PROGRAM F15_CaseControlCACData_ORG
VAR
	rtrigScanBarcode				: R_TRIG;
	fbScannerCtrl					: FB_SCANNER_CameraSelect;
	bScanCaseLabel				: BOOL;
	fbCaseLableEvaluation			: FB_SCANNER_Evaluation;

	rtrigSetCaseValidationOK			: R_TRIG;
	rtrigSetCaseValidationNOK		: R_TRIG;

	sCaseSerialCode				: T_CASE_Barcode;
	sFirstOuterInCase				: T_OUTER_Barcode;
	sLastOuterInCase				: T_OUTER_Barcode;
	sFirstPackSerialCode			: T_PACK_Barcode;
	sLastPackSerialCode				: T_PACK_Barcode;


	fbSequenceControl				: FB_SYSTEM_SeqControl;
	nSequenceStep				: INT;
	b00_Idle						: BOOL;
	b01_ScanLabel					: BOOL;
	b03_CreateFileName			: BOOL;
	b05_MoveCaseData				: BOOL;
	b08_WriteFSSFile				: BOOL;
	b10_CaseTraceValid			: BOOL;
	b18_CaseValid					: BOOL;
	b19_CaseInvalid				: BOOL;
	b20_Done						: BOOL;

	bDone						: BOOL;
	bBusy						: BOOL;
	tonScanTimeout					: TON;
	tonOverTime				: TON;

	rtrigCACData				: R_TRIG;
	tF15TimeExecution		: TIME;
	bTestSeq						: BOOL;
	sCACFileTemplate				: T_CAC_Filename;

	stValidateCACData				: ST_CAC_Data;
	fbMoveCaseData				: FB_CASE_ValidateAndMoveCACData;

	sPrintCaseContent				: STRING(255);

	fbPopulateCHMData				: FB_CHM_PopulateDataForFSS3;
	fbWriteCHMFile				: FB_CHM_WriteFSS3Files; (*Old system supporting FSS2 -> FB_CHM_WriteFSSFile;*)

	fbWriteCACToArchive 			: FB_CAC_WriteToArchive_v2;
	fbWriteCACToArchiveDB			: FB_CAC_WriteHierachyToDB;
	fbCaseStatusPulse				: TON;
	bCACValid					: BOOL;
	bCHMValid					: BOOL;


	fbMoveVerifiedCAC				: FB_CASE_MoveVerifiedCAC;
	fbMoveFailedCAC				: FB_CASE_MoveFailedCAC;

	fbCaseEfficiency				: FB_KPI_GenericEfficiency;
	fbCaseInspectionEfficiency		: FB_KPI_CaseEfficiency;
	(*fbCaseInspectionEfficiency		: FB_KPI_PACAN_CaseEfficiency;*)
	fbRejectCount					: CTU;
	nRejectActualCount				: INT;

	fbCaseValidationScanned			: FB_CTU32;
	fbCaseValidationCorrect			: FB_CTU32;
	fbCaseValidationNoCaseLabel		: FB_CTU32;
	fbCaseValidationCasePackerReject	: FB_CTU32;

	aLastCaseBarcodes				: ARRAY[1..cMAX_LAST_CASE_BARCODES] OF T_CASE_Barcode;
	fbAddVerifiedCaseBarcode		: FB_CASE_AddVerifiedCaseBarcode;

	fbCaseLevelCounter	: FB_KPI_CaseLevelCounter;
	tofCaseValidationCameraOFFDelay 	: TOF;

	fbFileWriteCACError				: FB_LOG_FileWriteError;
	fbFileWriteCHMError			: FB_LOG_FileWriteError;

END_VAR
(*
VAR CONSTANT
	sOptions						: ST_SCANNER_Options := (eScannerType := E_MV_440SR_FULL, nImageBuffer := 1, nExpectedResp := 1);
END_VAR*)
VAR // added by the converter: edge detectors and wires of the graphical bodies
    _w1 : ANY;
    _w2, _w3 : BOOL;
END_VAR

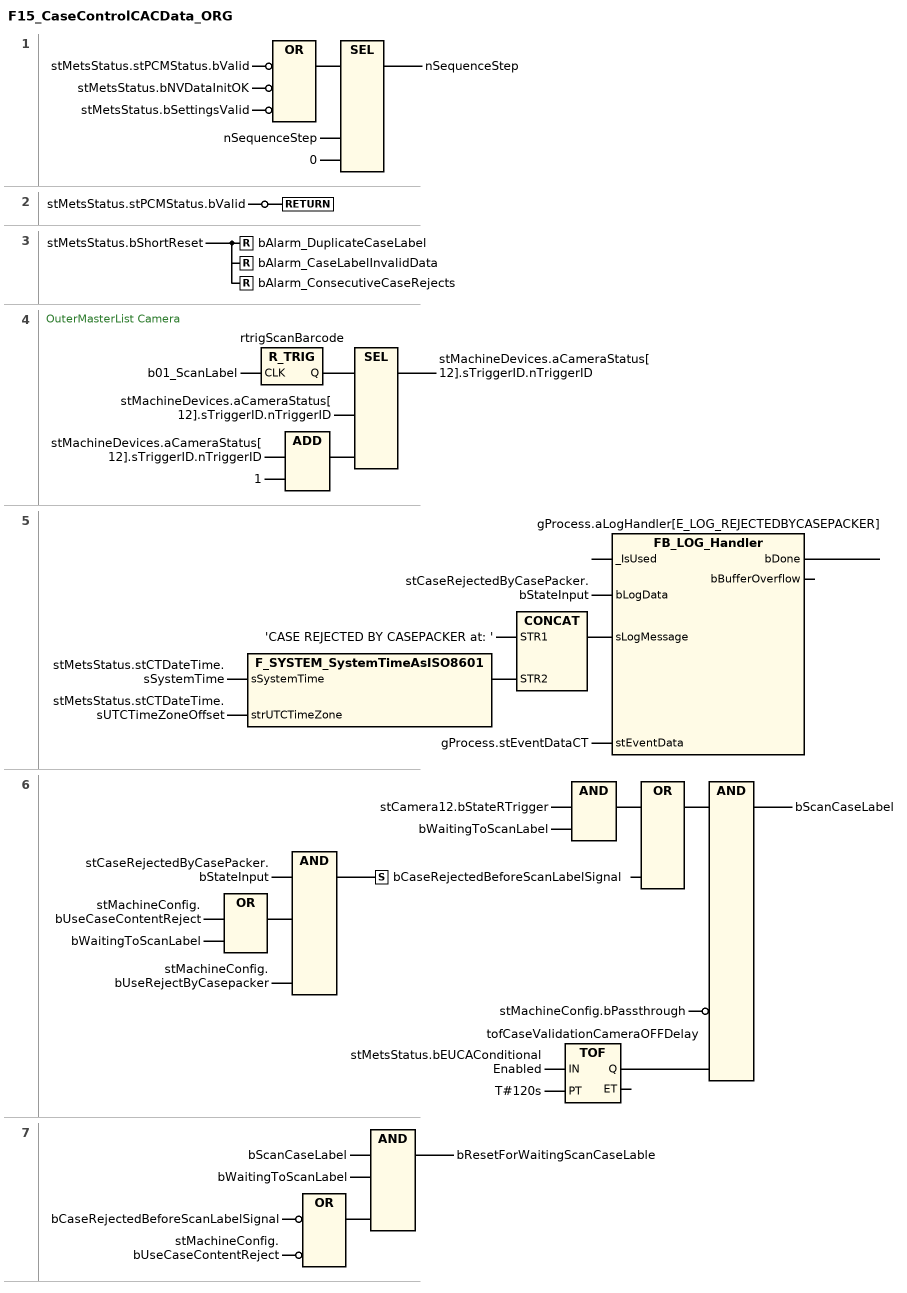
// NETWORK 1
nSequenceStep := SEL(NOT stMetsStatus.stPCMStatus.bValid OR NOT stMetsStatus.bNVDataInitOK OR NOT stMetsStatus.bSettingsValid, nSequenceStep, 0);

// NETWORK 2
IF NOT stMetsStatus.stPCMStatus.bValid THEN RETURN; END_IF

// NETWORK 3
bAlarm_DuplicateCaseLabel R= stMetsStatus.bShortReset;
bAlarm_CaseLabelInvalidData R= stMetsStatus.bShortReset;
bAlarm_ConsecutiveCaseRejects R= stMetsStatus.bShortReset;

// NETWORK 4
// OuterMasterList Camera
rtrigScanBarcode(CLK := b01_ScanLabel); // R_TRIG
stMachineDevices.aCameraStatus[12].sTriggerID.nTriggerID := SEL(rtrigScanBarcode.Q, stMachineDevices.aCameraStatus[12].sTriggerID.nTriggerID, stMachineDevices.aCameraStatus[12].sTriggerID.nTriggerID + 1);

// NETWORK 5
gProcess.aLogHandler[E_LOG_REJECTEDBYCASEPACKER](
    bLogData := stCaseRejectedByCasePacker.bStateInput,
    sLogMessage := CONCAT(STR1 := 'CASE REJECTED BY CASEPACKER at: ', STR2 := F_SYSTEM_SystemTimeAsISO8601(sSystemTime := stMetsStatus.stCTDateTime.sSystemTime, strUTCTimeZone := stMetsStatus.stCTDateTime.sUTCTimeZoneOffset)),
    stEventData := gProcess.stEventDataCT); // FB_LOG_Handler

// NETWORK 6
_w1 := stCaseRejectedByCasePacker.bStateInput AND (stMachineConfig.bUseCaseContentReject OR bWaitingToScanLabel) AND stMachineConfig.bUseRejectByCasepacker;
bCaseRejectedBeforeScanLabelSignal S= _w1;
tofCaseValidationCameraOFFDelay(IN := stMetsStatus.bEUCAConditionalEnabled, PT := T#120s); // TOF
bScanCaseLabel := (stCamera12.bStateRTrigger AND bWaitingToScanLabel OR _w1) AND NOT stMachineConfig.bPassthrough AND tofCaseValidationCameraOFFDelay.Q;

// NETWORK 7
bResetForWaitingScanCaseLable := bScanCaseLabel AND bWaitingToScanLabel AND (NOT bCaseRejectedBeforeScanLabelSignal OR NOT stMachineConfig.bUseCaseContentReject);

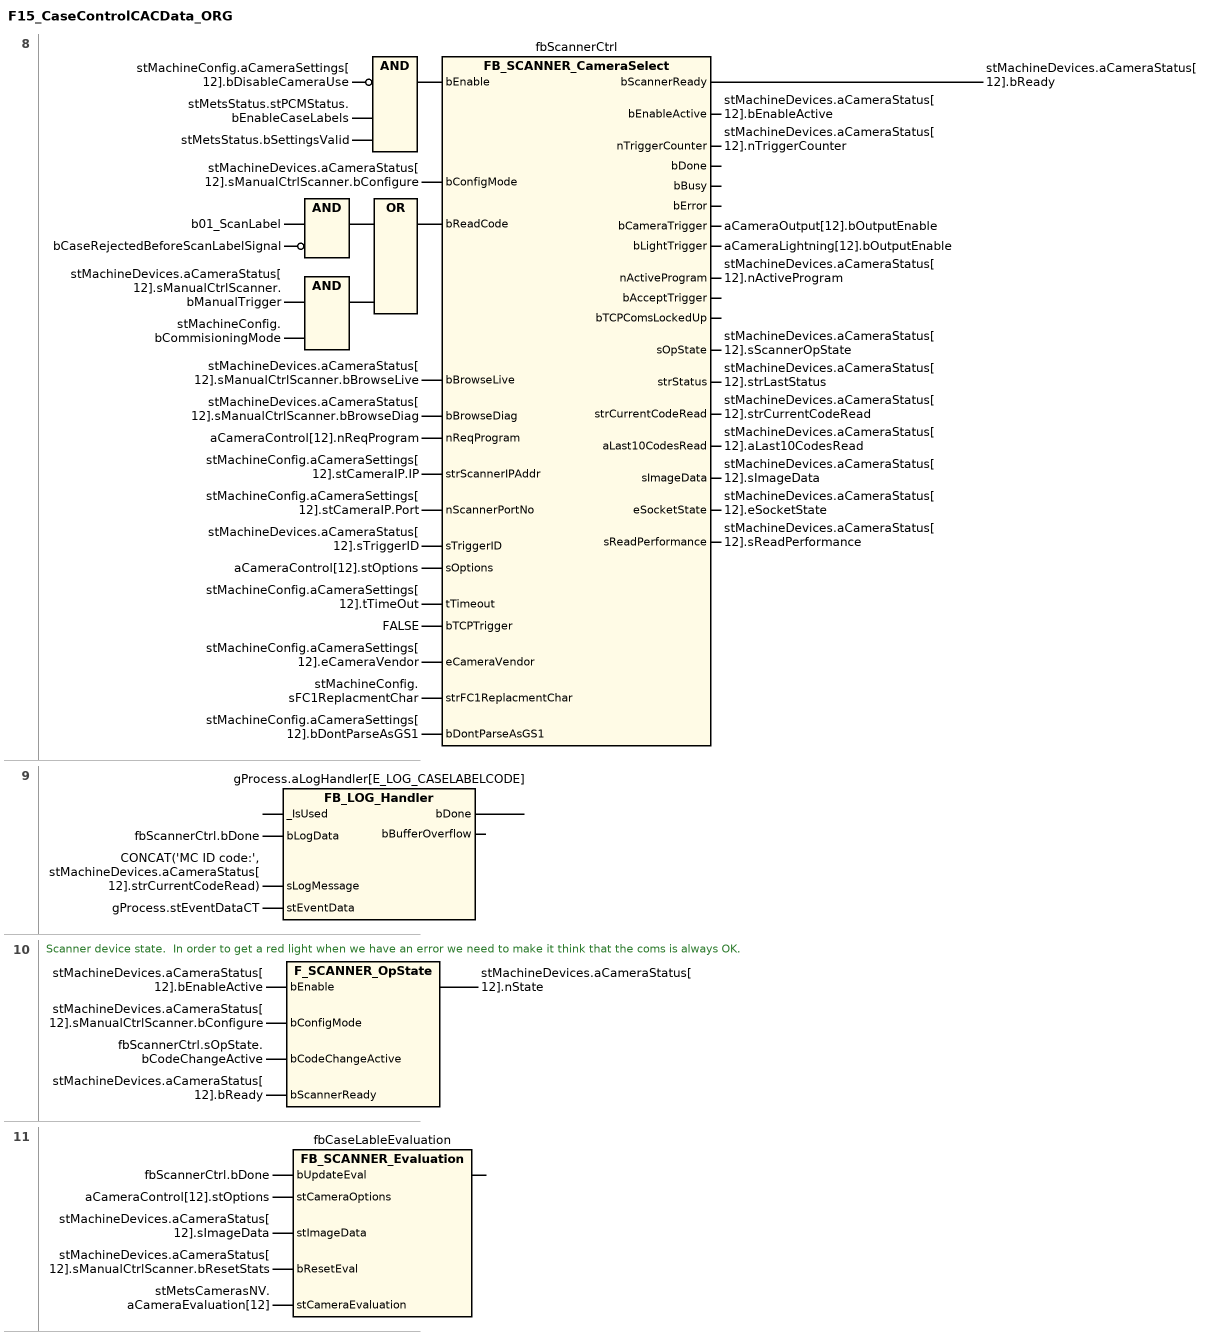
// NETWORK 8
fbScannerCtrl(
    bEnable := NOT stMachineConfig.aCameraSettings[12].bDisableCameraUse AND stMetsStatus.stPCMStatus.bEnableCaseLabels AND stMetsStatus.bSettingsValid,
    bConfigMode := stMachineDevices.aCameraStatus[12].sManualCtrlScanner.bConfigure,
    bReadCode := b01_ScanLabel AND NOT bCaseRejectedBeforeScanLabelSignal OR stMachineDevices.aCameraStatus[12].sManualCtrlScanner.bManualTrigger AND stMachineConfig.bCommisioningMode,
    bBrowseLive := stMachineDevices.aCameraStatus[12].sManualCtrlScanner.bBrowseLive,
    bBrowseDiag := stMachineDevices.aCameraStatus[12].sManualCtrlScanner.bBrowseDiag,
    nReqProgram := aCameraControl[12].nReqProgram,
    strScannerIPAddr := stMachineConfig.aCameraSettings[12].stCameraIP.IP,
    nScannerPortNo := stMachineConfig.aCameraSettings[12].stCameraIP.Port,
    sTriggerID := stMachineDevices.aCameraStatus[12].sTriggerID,
    sOptions := aCameraControl[12].stOptions,
    tTimeout := stMachineConfig.aCameraSettings[12].tTimeOut,
    bTCPTrigger := FALSE,
    eCameraVendor := stMachineConfig.aCameraSettings[12].eCameraVendor,
    strFC1ReplacmentChar := stMachineConfig.sFC1ReplacmentChar,
    bDontParseAsGS1 := stMachineConfig.aCameraSettings[12].bDontParseAsGS1,
    bEnableActive => stMachineDevices.aCameraStatus[12].bEnableActive,
    nTriggerCounter => stMachineDevices.aCameraStatus[12].nTriggerCounter,
    bCameraTrigger => aCameraOutput[12].bOutputEnable,
    bLightTrigger => aCameraLightning[12].bOutputEnable,
    nActiveProgram => stMachineDevices.aCameraStatus[12].nActiveProgram,
    sOpState => stMachineDevices.aCameraStatus[12].sScannerOpState,
    strStatus => stMachineDevices.aCameraStatus[12].strLastStatus,
    strCurrentCodeRead => stMachineDevices.aCameraStatus[12].strCurrentCodeRead,
    aLast10CodesRead => stMachineDevices.aCameraStatus[12].aLast10CodesRead,
    sImageData => stMachineDevices.aCameraStatus[12].sImageData,
    eSocketState => stMachineDevices.aCameraStatus[12].eSocketState,
    sReadPerformance => stMachineDevices.aCameraStatus[12].sReadPerformance); // FB_SCANNER_CameraSelect
stMachineDevices.aCameraStatus[12].bReady := fbScannerCtrl.bScannerReady;

// NETWORK 9
gProcess.aLogHandler[E_LOG_CASELABELCODE](
    bLogData := fbScannerCtrl.bDone,
    sLogMessage := CONCAT('MC ID code:', stMachineDevices.aCameraStatus[12].strCurrentCodeRead),
    stEventData := gProcess.stEventDataCT); // FB_LOG_Handler

// NETWORK 10
// Scanner device state.  In order to get a red light when we have an error we need to make it think that the coms is always OK.
stMachineDevices.aCameraStatus[12].nState := F_SCANNER_OpState(bEnable := stMachineDevices.aCameraStatus[12].bEnableActive, bConfigMode := stMachineDevices.aCameraStatus[12].sManualCtrlScanner.bConfigure, bCodeChangeActive := fbScannerCtrl.sOpState.bCodeChangeActive, bScannerReady := stMachineDevices.aCameraStatus[12].bReady);

// NETWORK 11
fbCaseLableEvaluation(
    bUpdateEval := fbScannerCtrl.bDone,
    stCameraOptions := aCameraControl[12].stOptions,
    stImageData := stMachineDevices.aCameraStatus[12].sImageData,
    bResetEval := stMachineDevices.aCameraStatus[12].sManualCtrlScanner.bResetStats,
    stCameraEvaluation := stMetsCamerasNV.aCameraEvaluation[12]); // FB_SCANNER_Evaluation

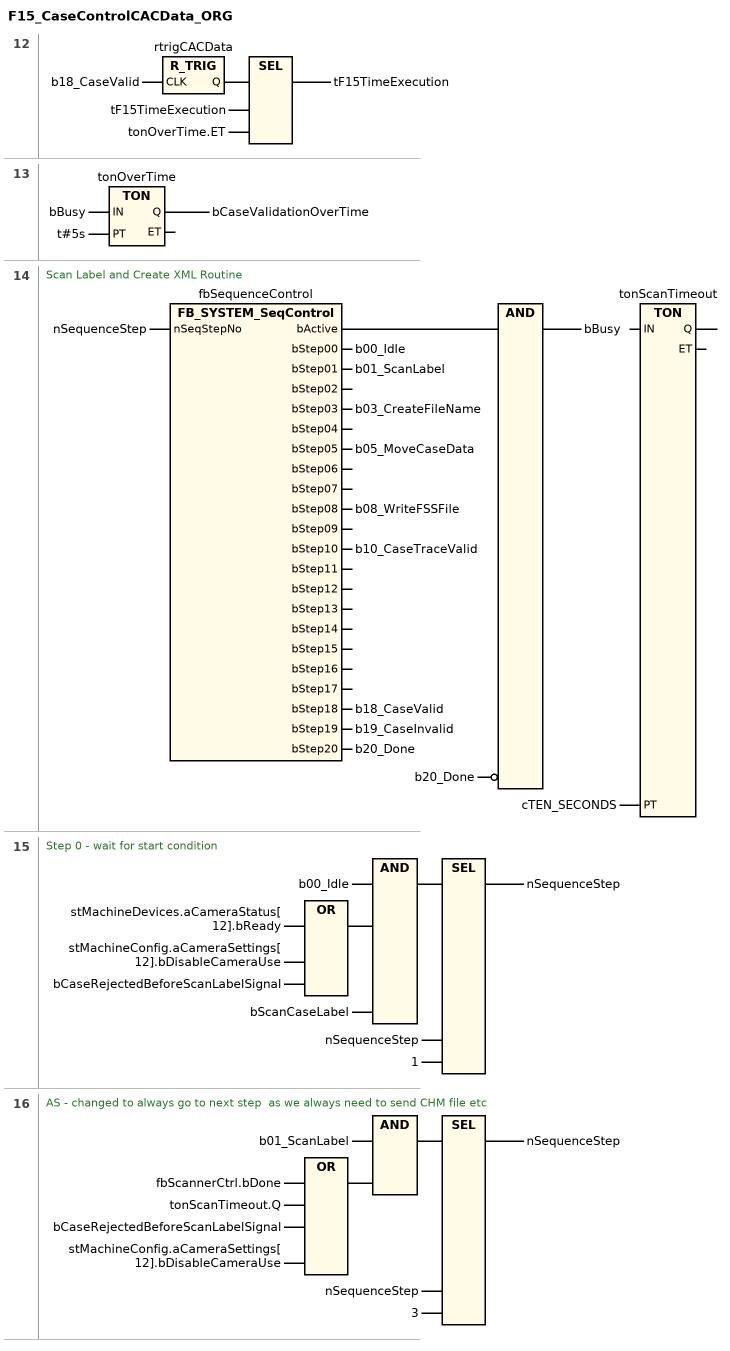
// NETWORK 12
rtrigCACData(CLK := b18_CaseValid); // R_TRIG
tF15TimeExecution := SEL(rtrigCACData.Q, tF15TimeExecution, tonOverTime.ET);

// NETWORK 13
tonOverTime(IN := bBusy, PT := t#5s); // TON
bCaseValidationOverTime := tonOverTime.Q;

// NETWORK 14
// 					Scan Label and Create XML Routine
//
//
//
fbSequenceControl(
    nSeqStepNo := nSequenceStep,
    bStep00 => b00_Idle,
    bStep01 => b01_ScanLabel,
    bStep03 => b03_CreateFileName,
    bStep05 => b05_MoveCaseData,
    bStep08 => b08_WriteFSSFile,
    bStep10 => b10_CaseTraceValid,
    bStep18 => b18_CaseValid,
    bStep19 => b19_CaseInvalid,
    bStep20 => b20_Done); // FB_SYSTEM_SeqControl
_w2 := fbSequenceControl.bActive AND NOT b20_Done;
bBusy := _w2;
tonScanTimeout(IN := _w2, PT := cTEN_SECONDS); // TON

// NETWORK 15
// 					Step 0 - wait for start condition
//
//
nSequenceStep := SEL(b00_Idle AND (stMachineDevices.aCameraStatus[12].bReady OR stMachineConfig.aCameraSettings[12].bDisableCameraUse OR bCaseRejectedBeforeScanLabelSignal) AND bScanCaseLabel, nSequenceStep, 1);

// NETWORK 16
// 					AS - changed to always go to next step  as we always need to send CHM file etc
//
//
nSequenceStep := SEL(b01_ScanLabel AND (fbScannerCtrl.bDone OR tonScanTimeout.Q OR bCaseRejectedBeforeScanLabelSignal OR stMachineConfig.aCameraSettings[12].bDisableCameraUse), nSequenceStep, 3);

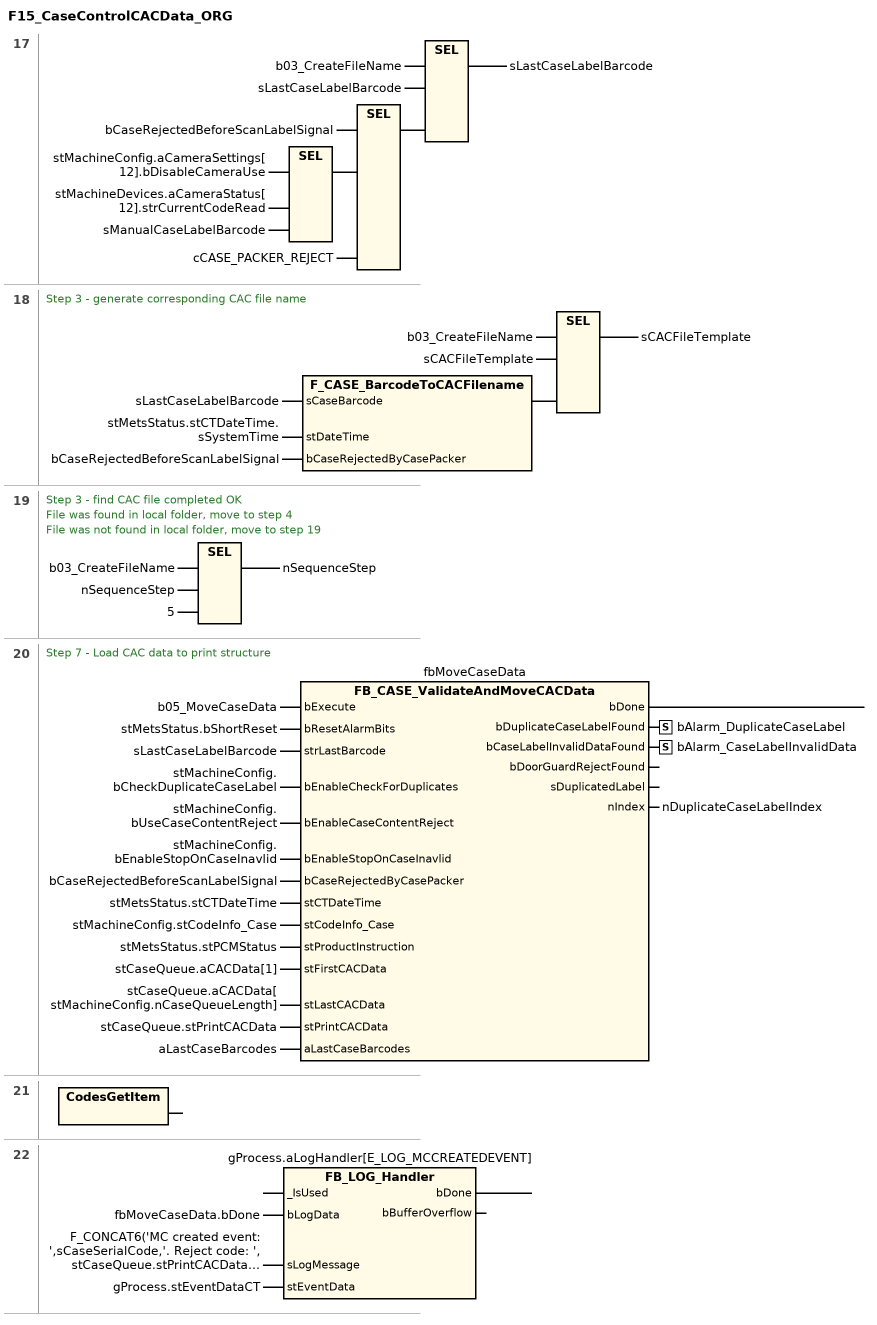
// NETWORK 17
sLastCaseLabelBarcode := SEL(b03_CreateFileName, sLastCaseLabelBarcode, SEL(bCaseRejectedBeforeScanLabelSignal, SEL(stMachineConfig.aCameraSettings[12].bDisableCameraUse, stMachineDevices.aCameraStatus[12].strCurrentCodeRead, sManualCaseLabelBarcode), cCASE_PACKER_REJECT));

// NETWORK 18
// Step 3 - generate corresponding CAC file name
sCACFileTemplate := SEL(b03_CreateFileName, sCACFileTemplate, F_CASE_BarcodeToCACFilename(sCaseBarcode := sLastCaseLabelBarcode, stDateTime := stMetsStatus.stCTDateTime.sSystemTime, bCaseRejectedByCasePacker := bCaseRejectedBeforeScanLabelSignal));

// NETWORK 19
// 					Step 3 - find CAC file completed OK
// File was found in local folder, move to step 4
// File was not found in local folder, move to step 19
//
nSequenceStep := SEL(b03_CreateFileName, nSequenceStep, 5);

// NETWORK 20
// Step 7 - Load CAC data to print structure
fbMoveCaseData(
    bExecute := b05_MoveCaseData,
    bResetAlarmBits := stMetsStatus.bShortReset,
    strLastBarcode := sLastCaseLabelBarcode,
    bEnableCheckForDuplicates := stMachineConfig.bCheckDuplicateCaseLabel,
    bEnableCaseContentReject := stMachineConfig.bUseCaseContentReject,
    bEnableStopOnCaseInavlid := stMachineConfig.bEnableStopOnCaseInavlid,
    bCaseRejectedByCasePacker := bCaseRejectedBeforeScanLabelSignal,
    stCTDateTime := stMetsStatus.stCTDateTime,
    stCodeInfo_Case := stMachineConfig.stCodeInfo_Case,
    stProductInstruction := stMetsStatus.stPCMStatus,
    stFirstCACData := stCaseQueue.aCACData[1],
    stLastCACData := stCaseQueue.aCACData[stMachineConfig.nCaseQueueLength],
    stPrintCACData := stCaseQueue.stPrintCACData,
    aLastCaseBarcodes := aLastCaseBarcodes,
    nIndex => nDuplicateCaseLabelIndex); // FB_CASE_ValidateAndMoveCACData
bAlarm_DuplicateCaseLabel S= fbMoveCaseData.bDuplicateCaseLabelFound;
bAlarm_CaseLabelInvalidData S= fbMoveCaseData.bCaseLabelInvalidDataFound;

// NETWORK 21
CodesGetItem();

// NETWORK 22
gProcess.aLogHandler[E_LOG_MCCREATEDEVENT](
    bLogData := fbMoveCaseData.bDone,
    sLogMessage := F_CONCAT6('MC created event: ',sCaseSerialCode,'. Reject code: ', stCaseQueue.stPrintCACData.CaseRejectCode,', with case content: ', sPrintCaseContent),
    stEventData := gProcess.stEventDataCT); // FB_LOG_Handler

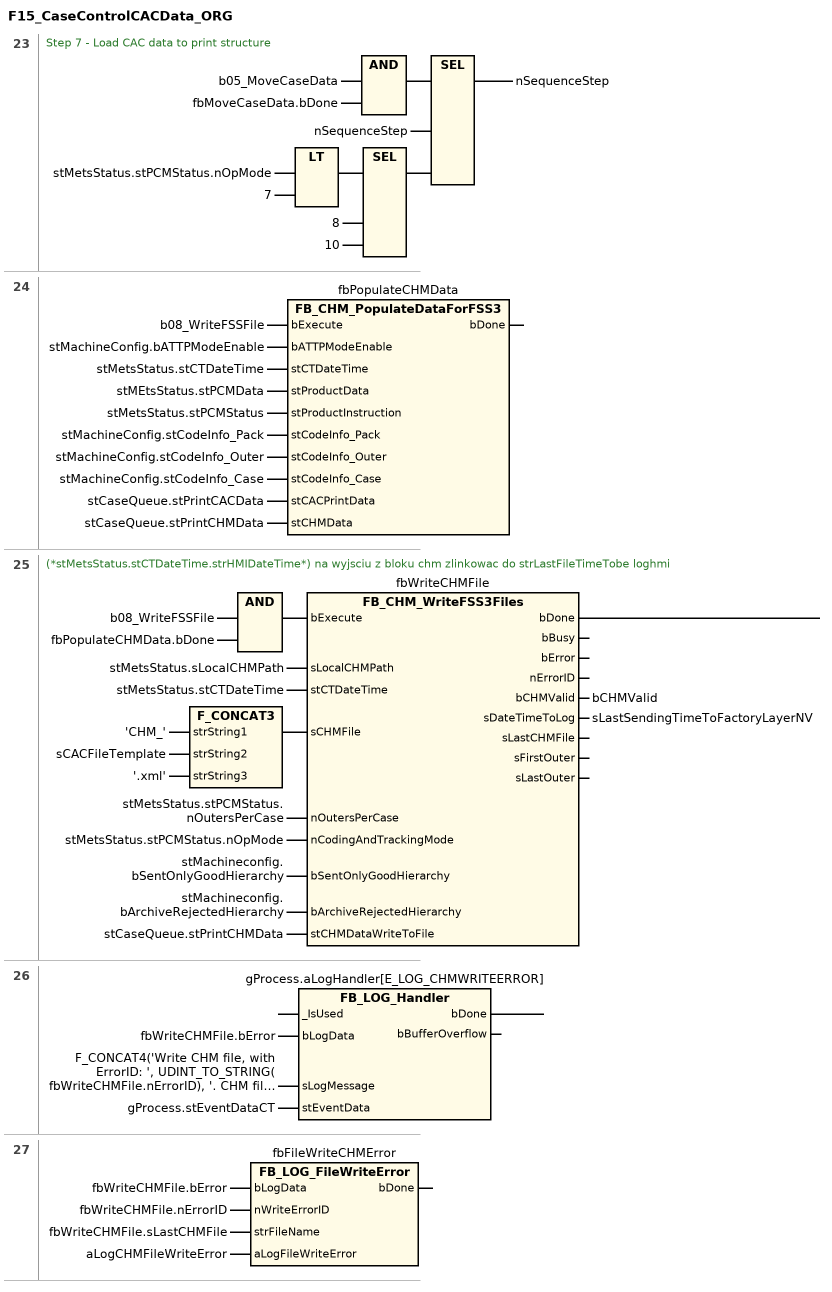
// NETWORK 23
// 					Step 7 - Load CAC data to print structure
//
//
nSequenceStep := SEL(b05_MoveCaseData AND fbMoveCaseData.bDone, nSequenceStep, SEL(stMetsStatus.stPCMStatus.nOpMode < 7, 8, 10));

// NETWORK 24
fbPopulateCHMData(
    bExecute := b08_WriteFSSFile,
    bATTPModeEnable := stMachineConfig.bATTPModeEnable,
    stCTDateTime := stMetsStatus.stCTDateTime,
    stProductData := stMEtsStatus.stPCMData,
    stProductInstruction := stMetsStatus.stPCMStatus,
    stCodeInfo_Pack := stMachineConfig.stCodeInfo_Pack,
    stCodeInfo_Outer := stMachineConfig.stCodeInfo_Outer,
    stCodeInfo_Case := stMachineConfig.stCodeInfo_Case,
    stCACPrintData := stCaseQueue.stPrintCACData,
    stCHMData := stCaseQueue.stPrintCHMData); // FB_CHM_PopulateDataForFSS3

// NETWORK 25
// (*stMetsStatus.stCTDateTime.strHMIDateTime*) na wyjsciu z bloku chm zlinkowac do strLastFileTimeTobe loghmi
fbWriteCHMFile(
    bExecute := b08_WriteFSSFile AND fbPopulateCHMData.bDone,
    sLocalCHMPath := stMetsStatus.sLocalCHMPath,
    stCTDateTime := stMetsStatus.stCTDateTime,
    sCHMFile := F_CONCAT3(strString1 := 'CHM_', strString2 := sCACFileTemplate, strString3 := '.xml'),
    nOutersPerCase := stMetsStatus.stPCMStatus.nOutersPerCase,
    nCodingAndTrackingMode := stMetsStatus.stPCMStatus.nOpMode,
    bSentOnlyGoodHierarchy := stMachineconfig.bSentOnlyGoodHierarchy,
    bArchiveRejectedHierarchy := stMachineconfig.bArchiveRejectedHierarchy,
    stCHMDataWriteToFile := stCaseQueue.stPrintCHMData,
    bCHMValid => bCHMValid,
    sDateTimeToLog => sLastSendingTimeToFactoryLayerNV); // FB_CHM_WriteFSS3Files

// NETWORK 26
gProcess.aLogHandler[E_LOG_CHMWRITEERROR](
    bLogData := fbWriteCHMFile.bError,
    sLogMessage := F_CONCAT4('Write CHM file, with ErrorID: ', UDINT_TO_STRING(fbWriteCHMFile.nErrorID), '. CHM file name: ', fbWriteCHMFile.sCHMFile),
    stEventData := gProcess.stEventDataCT); // FB_LOG_Handler

// NETWORK 27
fbFileWriteCHMError(
    bLogData := fbWriteCHMFile.bError,
    nWriteErrorID := fbWriteCHMFile.nErrorID,
    strFileName := fbWriteCHMFile.sLastCHMFile,
    aLogFileWriteError := aLogCHMFileWriteError); // FB_LOG_FileWriteError

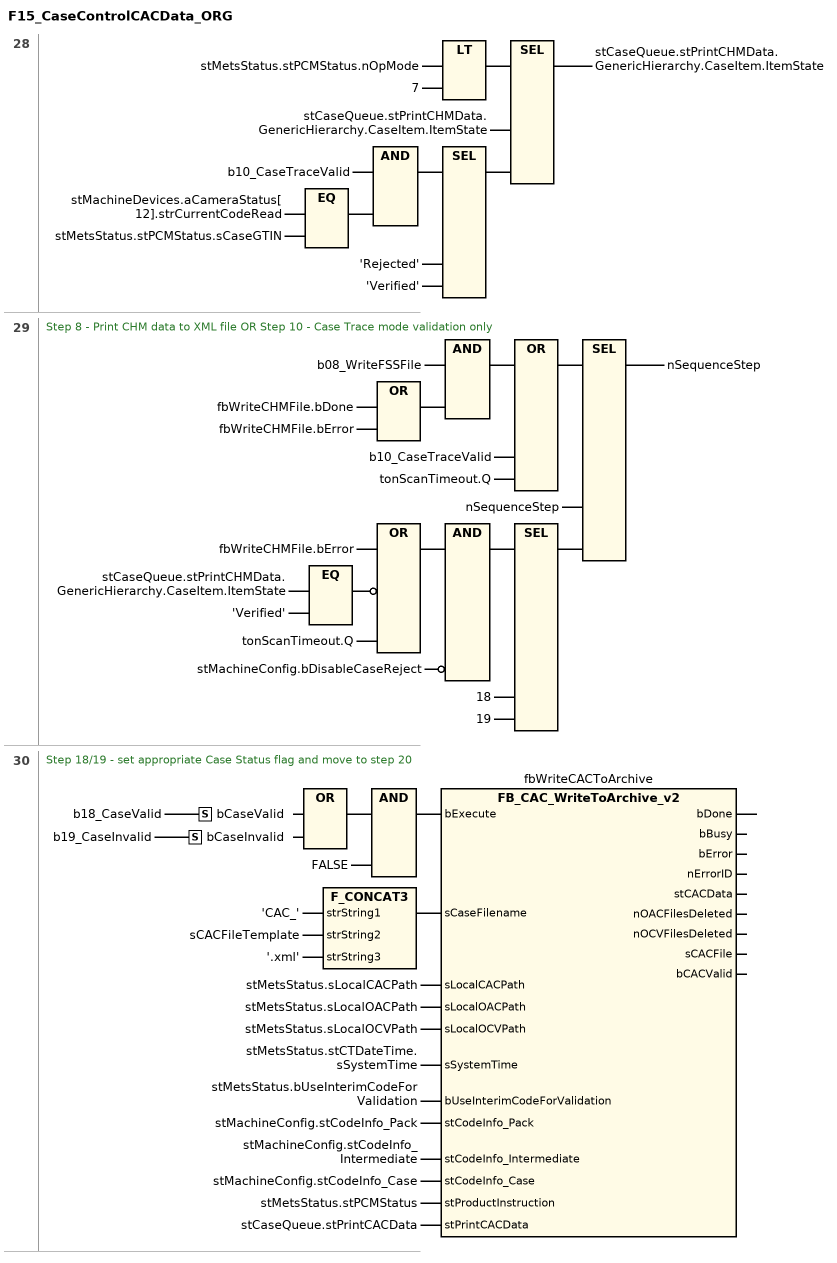
// NETWORK 28
stCaseQueue.stPrintCHMData.GenericHierarchy.CaseItem.ItemState := SEL(stMetsStatus.stPCMStatus.nOpMode < 7, stCaseQueue.stPrintCHMData.GenericHierarchy.CaseItem.ItemState, SEL(b10_CaseTraceValid AND stMachineDevices.aCameraStatus[12].strCurrentCodeRead = stMetsStatus.stPCMStatus.sCaseGTIN, 'Rejected', 'Verified'));

// NETWORK 29
// Step 8 - Print CHM data to XML file OR Step 10 - Case Trace mode validation only
nSequenceStep := SEL(b08_WriteFSSFile AND (fbWriteCHMFile.bDone OR fbWriteCHMFile.bError) OR b10_CaseTraceValid OR tonScanTimeout.Q, nSequenceStep, SEL((fbWriteCHMFile.bError OR NOT (stCaseQueue.stPrintCHMData.GenericHierarchy.CaseItem.ItemState = 'Verified') OR tonScanTimeout.Q) AND NOT stMachineConfig.bDisableCaseReject, 18, 19));

// NETWORK 30
// Step 18/19 - set appropriate Case Status flag and move to step 20
bCaseValid S= b18_CaseValid;
bCaseInvalid S= b19_CaseInvalid;
fbWriteCACToArchive(
    bExecute := (b18_CaseValid OR b19_CaseInvalid) AND FALSE,
    sCaseFilename := F_CONCAT3(strString1 := 'CAC_', strString2 := sCACFileTemplate, strString3 := '.xml'),
    sLocalCACPath := stMetsStatus.sLocalCACPath,
    sLocalOACPath := stMetsStatus.sLocalOACPath,
    sLocalOCVPath := stMetsStatus.sLocalOCVPath,
    sSystemTime := stMetsStatus.stCTDateTime.sSystemTime,
    bUseInterimCodeForValidation := stMetsStatus.bUseInterimCodeForValidation,
    stCodeInfo_Pack := stMachineConfig.stCodeInfo_Pack,
    stCodeInfo_Intermediate := stMachineConfig.stCodeInfo_Intermediate,
    stCodeInfo_Case := stMachineConfig.stCodeInfo_Case,
    stProductInstruction := stMetsStatus.stPCMStatus,
    stPrintCACData := stCaseQueue.stPrintCACData); // FB_CAC_WriteToArchive_v2

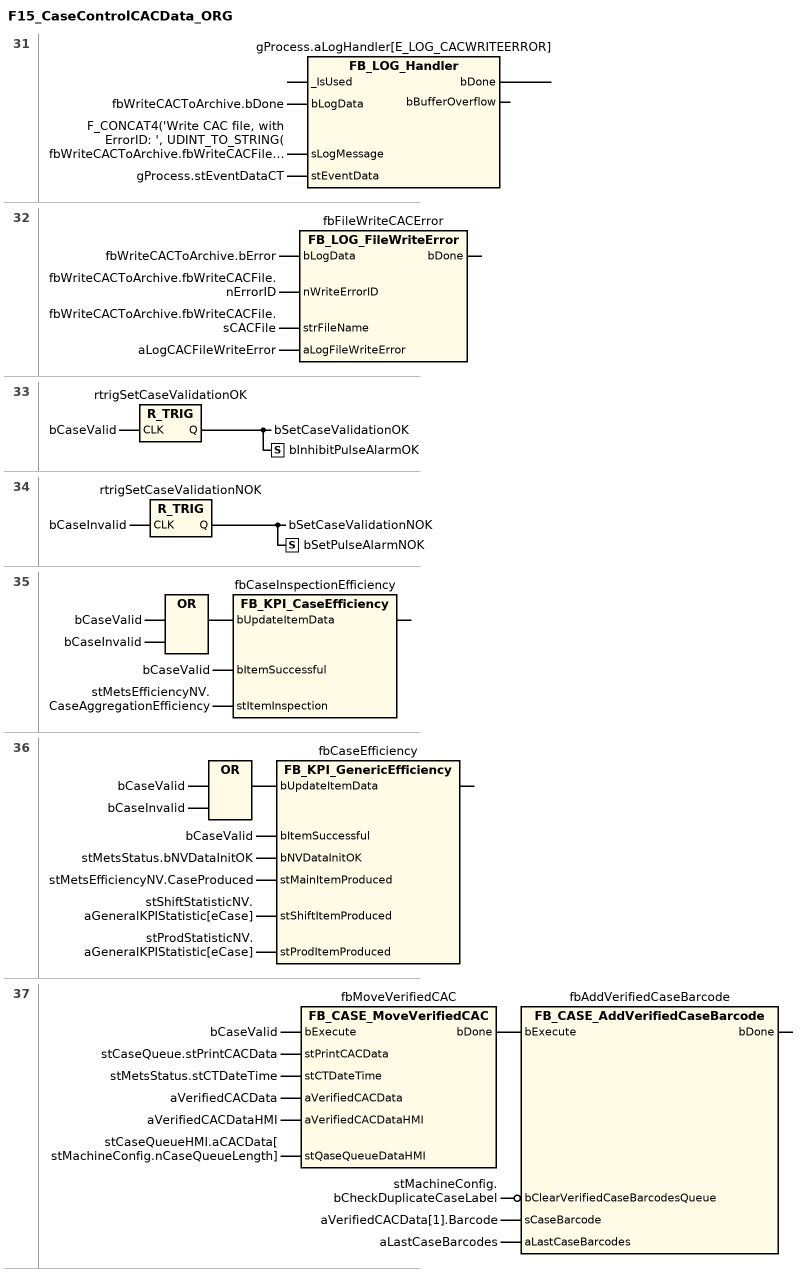
// NETWORK 31
gProcess.aLogHandler[E_LOG_CACWRITEERROR](
    bLogData := fbWriteCACToArchive.bDone,
    sLogMessage := F_CONCAT4('Write CAC file, with ErrorID: ', UDINT_TO_STRING(fbWriteCACToArchive.fbWriteCACFile.nErrorID), '. CAC file name: ', fbWriteCACToArchive.fbWriteCACFile.sCACFile),
    stEventData := gProcess.stEventDataCT); // FB_LOG_Handler

// NETWORK 32
fbFileWriteCACError(
    bLogData := fbWriteCACToArchive.bError,
    nWriteErrorID := fbWriteCACToArchive.fbWriteCACFile.nErrorID,
    strFileName := fbWriteCACToArchive.fbWriteCACFile.sCACFile,
    aLogFileWriteError := aLogCACFileWriteError); // FB_LOG_FileWriteError

// NETWORK 33
rtrigSetCaseValidationOK(CLK := bCaseValid); // R_TRIG
bSetCaseValidationOK := rtrigSetCaseValidationOK.Q;
bInhibitPulseAlarmOK S= rtrigSetCaseValidationOK.Q;

// NETWORK 34
rtrigSetCaseValidationNOK(CLK := bCaseInvalid); // R_TRIG
bSetCaseValidationNOK := rtrigSetCaseValidationNOK.Q;
bSetPulseAlarmNOK S= rtrigSetCaseValidationNOK.Q;

// NETWORK 35
fbCaseInspectionEfficiency(
    bUpdateItemData := bCaseValid OR bCaseInvalid,
    bItemSuccessful := bCaseValid,
    stItemInspection := stMetsEfficiencyNV.CaseAggregationEfficiency); // FB_KPI_CaseEfficiency

// NETWORK 36
fbCaseEfficiency(
    bUpdateItemData := bCaseValid OR bCaseInvalid,
    bItemSuccessful := bCaseValid,
    bNVDataInitOK := stMetsStatus.bNVDataInitOK,
    stMainItemProduced := stMetsEfficiencyNV.CaseProduced,
    stShiftItemProduced := stShiftStatisticNV.aGeneralKPIStatistic[eCase],
    stProdItemProduced := stProdStatisticNV.aGeneralKPIStatistic[eCase]); // FB_KPI_GenericEfficiency

// NETWORK 37
fbMoveVerifiedCAC(
    bExecute := bCaseValid,
    stPrintCACData := stCaseQueue.stPrintCACData,
    stCTDateTime := stMetsStatus.stCTDateTime,
    aVerifiedCACData := aVerifiedCACData,
    aVerifiedCACDataHMI := aVerifiedCACDataHMI,
    stQaseQueueDataHMI := stCaseQueueHMI.aCACData[stMachineConfig.nCaseQueueLength]); // FB_CASE_MoveVerifiedCAC
fbAddVerifiedCaseBarcode(
    bExecute := fbMoveVerifiedCAC.bDone,
    bClearVerifiedCaseBarcodesQueue := NOT stMachineConfig.bCheckDuplicateCaseLabel,
    sCaseBarcode := aVerifiedCACData[1].Barcode,
    aLastCaseBarcodes := aLastCaseBarcodes); // FB_CASE_AddVerifiedCaseBarcode

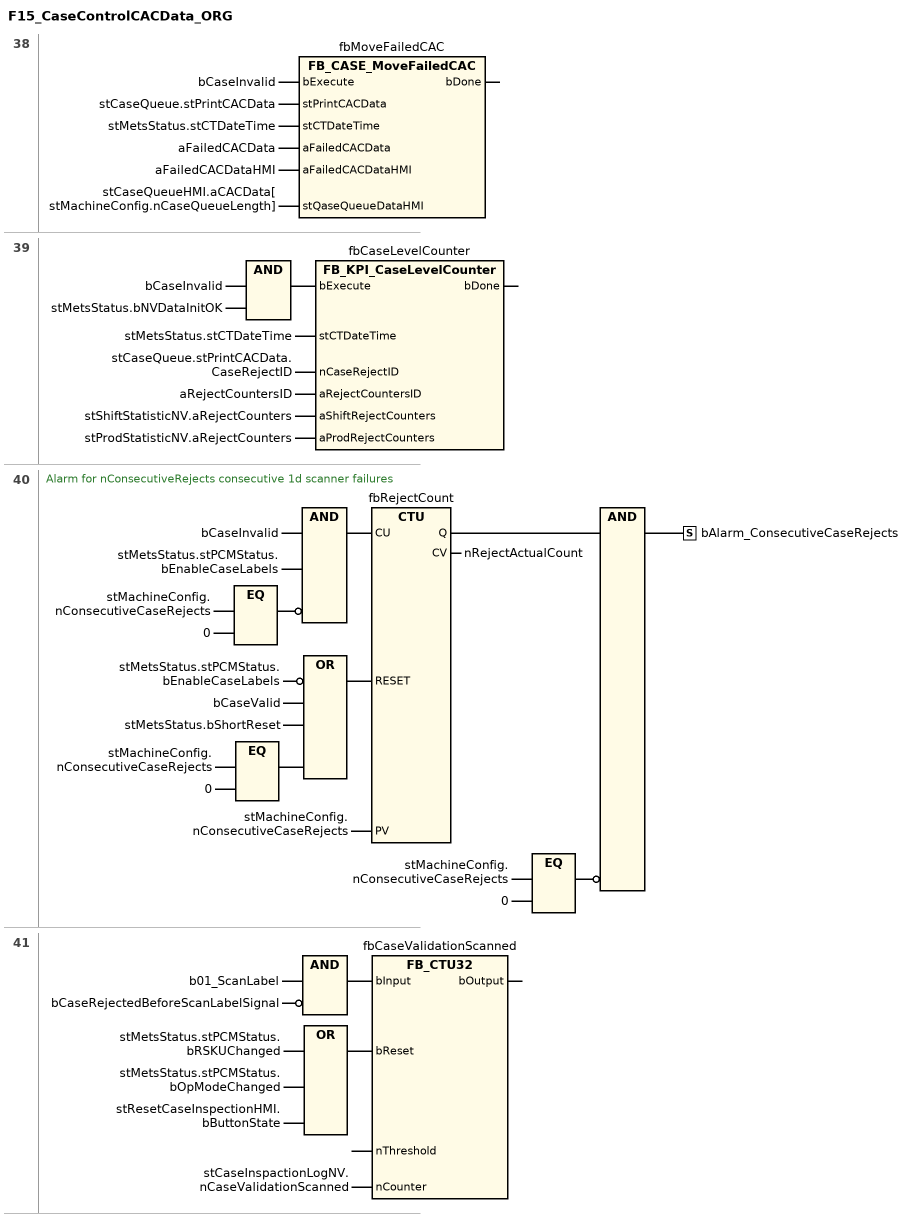
// NETWORK 38
fbMoveFailedCAC(
    bExecute := bCaseInvalid,
    stPrintCACData := stCaseQueue.stPrintCACData,
    stCTDateTime := stMetsStatus.stCTDateTime,
    aFailedCACData := aFailedCACData,
    aFailedCACDataHMI := aFailedCACDataHMI,
    stQaseQueueDataHMI := stCaseQueueHMI.aCACData[stMachineConfig.nCaseQueueLength]); // FB_CASE_MoveFailedCAC

// NETWORK 39
fbCaseLevelCounter(
    bExecute := bCaseInvalid AND stMetsStatus.bNVDataInitOK,
    stCTDateTime := stMetsStatus.stCTDateTime,
    nCaseRejectID := stCaseQueue.stPrintCACData.CaseRejectID,
    aRejectCountersID := aRejectCountersID,
    aShiftRejectCounters := stShiftStatisticNV.aRejectCounters,
    aProdRejectCounters := stProdStatisticNV.aRejectCounters); // FB_KPI_CaseLevelCounter

// NETWORK 40
// Alarm for nConsecutiveRejects consecutive 1d scanner failures
fbRejectCount(
    CU := bCaseInvalid AND stMetsStatus.stPCMStatus.bEnableCaseLabels AND NOT (stMachineConfig.nConsecutiveCaseRejects = 0),
    RESET := NOT stMetsStatus.stPCMStatus.bEnableCaseLabels OR bCaseValid OR stMetsStatus.bShortReset OR stMachineConfig.nConsecutiveCaseRejects = 0,
    PV := stMachineConfig.nConsecutiveCaseRejects,
    CV => nRejectActualCount); // CTU
bAlarm_ConsecutiveCaseRejects S= fbRejectCount.Q AND NOT (stMachineConfig.nConsecutiveCaseRejects = 0);

// NETWORK 41
fbCaseValidationScanned(
    bInput := b01_ScanLabel AND NOT bCaseRejectedBeforeScanLabelSignal,
    bReset := stMetsStatus.stPCMStatus.bRSKUChanged OR stMetsStatus.stPCMStatus.bOpModeChanged OR stResetCaseInspectionHMI.bButtonState,
    nCounter := stCaseInspactionLogNV.nCaseValidationScanned); // FB_CTU32

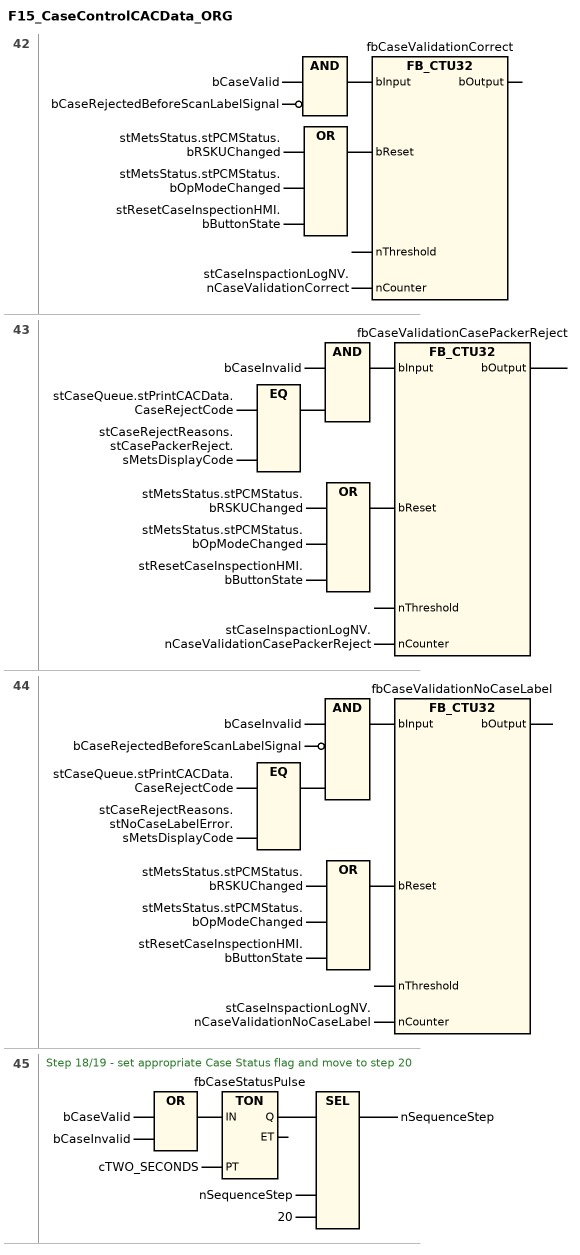
// NETWORK 42
fbCaseValidationCorrect(
    bInput := bCaseValid AND NOT bCaseRejectedBeforeScanLabelSignal,
    bReset := stMetsStatus.stPCMStatus.bRSKUChanged OR stMetsStatus.stPCMStatus.bOpModeChanged OR stResetCaseInspectionHMI.bButtonState,
    nCounter := stCaseInspactionLogNV.nCaseValidationCorrect); // FB_CTU32

// NETWORK 43
fbCaseValidationCasePackerReject(
    bInput := bCaseInvalid AND stCaseQueue.stPrintCACData.CaseRejectCode = stCaseRejectReasons.stCasePackerReject.sMetsDisplayCode,
    bReset := stMetsStatus.stPCMStatus.bRSKUChanged OR stMetsStatus.stPCMStatus.bOpModeChanged OR stResetCaseInspectionHMI.bButtonState,
    nCounter := stCaseInspactionLogNV.nCaseValidationCasePackerReject); // FB_CTU32

// NETWORK 44
fbCaseValidationNoCaseLabel(
    bInput := bCaseInvalid AND NOT bCaseRejectedBeforeScanLabelSignal AND stCaseQueue.stPrintCACData.CaseRejectCode = stCaseRejectReasons.stNoCaseLabelError.sMetsDisplayCode,
    bReset := stMetsStatus.stPCMStatus.bRSKUChanged OR stMetsStatus.stPCMStatus.bOpModeChanged OR stResetCaseInspectionHMI.bButtonState,
    nCounter := stCaseInspactionLogNV.nCaseValidationNoCaseLabel); // FB_CTU32

// NETWORK 45
// Step 18/19 - set appropriate Case Status flag and move to step 20
fbCaseStatusPulse(IN := bCaseValid OR bCaseInvalid, PT := cTWO_SECONDS); // TON
nSequenceStep := SEL(fbCaseStatusPulse.Q, nSequenceStep, 20);

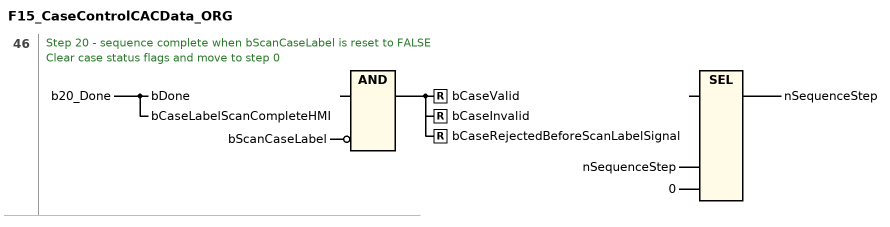
// NETWORK 46
// 					Step 20 - sequence complete when bScanCaseLabel is reset to FALSE
// Clear case status flags and move to step 0
//
bDone := b20_Done;
bCaseLabelScanCompleteHMI := b20_Done;
_w3 := b20_Done AND NOT bScanCaseLabel;
bCaseValid R= _w3;
bCaseInvalid R= _w3;
bCaseRejectedBeforeScanLabelSignal R= _w3;
nSequenceStep := SEL(_w3, nSequenceStep, 0);

ACTION CodesGetItem:
IF stMetsStatus.stPCMStatus.nOutersPerCase > 0 AND stMetsStatus.stPCMStatus.nPacksPerOuter > 0 THEN

	sCaseSerialCode := F_CODE_GetItem(stCaseQueue.stPrintCACData.Barcode, eCodeAIType.SerialCode, stMachineConfig.stCodeInfo_Case);
	sFirstOuterInCase := F_CODE_GetItem(stCaseQueue.stPrintCACData.Outer[1].Barcode, eCodeAIType.SerialCode, stMachineConfig.stCodeInfo_Outer);
	sLastOuterInCase := F_CODE_GetItem(stCaseQueue.stPrintCACData.Outer[stMetsStatus.stPCMStatus.nOutersPerCase].Barcode, eCodeAIType.SerialCode, stMachineConfig.stCodeInfo_Outer);
	sFirstPackSerialCode := F_CODE_GetItem(stCaseQueue.stPrintCACData.Outer[1].PackCode[1], eCodeAIType.SerialCode, stMachineConfig.stCodeInfo_Pack);
	sLastPackSerialCode := F_CODE_GetItem(stCaseQueue.stPrintCACData.Outer[stMetsStatus.stPCMStatus.nOutersPerCase].PackCode[stMetsStatus.stPCMStatus.nPacksPerOuter], eCodeAIType.SerialCode, stMachineConfig.stCodeInfo_Pack);

	sFirstOuterInCase	:= RIGHT(sFirstOuterInCase,7);
	sLastOuterInCase	:= RIGHT(sLastOuterInCase,7);
	sFirstPackSerialCode	:= RIGHT(sFirstPackSerialCode,7);
	sLastPackSerialCode	:= RIGHT(sLastPackSerialCode,7);

	sPrintCaseContent  := F_CONCAT9('Init OUT ID [',sFirstOuterInCase, '] ; Last OUT ID [', sLastOuterInCase,  '] ; Init PK ID [',sFirstPackSerialCode, '] ; Last PK ID [', sLastPackSerialCode,']');
END_IF
END_ACTION

END_PROGRAM

(* stored: Version 1.1.0.1
   POU F15_CaseControlCACData_ORG: Id {048f1acd-90d8-44f9-bb12-acc3378d5fd2}, SpecialFunc None
   Action CodesGetItem: Id {f9a4654e-b2d6-4757-a308-e8c919983a19} *)
